FUNCTION_BLOCK ChangeDetect (* Ground-truth reference: fires CHG only when the REAL input value actually changed *)
  (* Standard: 61499-2; Description: Educational reference, ported for the Meisterschulen am Ostbahnhof IEC 61499 training repository. Original design (c) nxtControl GmbH, from the UniversalAutomation.org 'IEC 61499: primer course' curriculum exercise Final.sln (also present in the LiftingLuggage_*.sln/Starter.sln exercises), IEC61499/ChangeDetect.fbt - included here under the same educational-use terms as the rest of that curriculum. This port: Copyright (c) 2026 Meisterschulen am Ostbahnhof, EPL-2.0, https://www.eclipse.org/legal/epl-2.0/ *)
  (* Version 0.0, 2016-05-28, Andrei, nxtControl GmbH, Original EAE/nxtControl design (Template), source: Final.sln (identical copies in LiftingLuggage_*.sln, Starter.sln) *)
  (* Version 1.0, 2026-09-03, Franz Höpfinger, Meisterschulen am Ostbahnhof, Ported from EAE/nxtControl format (LibraryElement.dtd, ST as an attribute with escapes) to 4diac's FBType XSD (ST as CDATA). Interface, ECC, and both algorithms otherwise unchanged. Part of the CylinderH continuous-simulation reference - see ContinuousCylinderSimulation.md *)
  PACKAGE Meins::DesingPatterns::ContinuousCylinderSimulation;
  (* Documentation:
  Ground-truth reference, not a Vyatkin Module 6 slide pattern. Simple REAL change-detection filter, ported as-is from the UniversalAutomation.org "IEC 61499: primer course" curriculum (Final.sln, IEC61499/ChangeDetect.fbt, original format: EAE/nxtControl LibraryElement.dtd). Used by CylinderHCore.fbt in this folder to throttle the integrator's continuous out value down to only the moments it actually changes, before reporting the cylinder's Position onward.
  *)
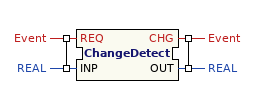
  EVENT_INPUT
    REQ WITH INP; (* Normal Execution Request *)
  END_EVENT
  EVENT_OUTPUT
    CHG WITH OUT; (* Execution Confirmation: fired every REQ, but only carries a new value on an actual change *)
  END_EVENT
  VAR_INPUT
    INP : REAL;
  END_VAR
  VAR_OUTPUT
    OUT : REAL;
  END_VAR
  VAR
    PREV : REAL; (* Value seen on the previous REQ *)
  END_VAR
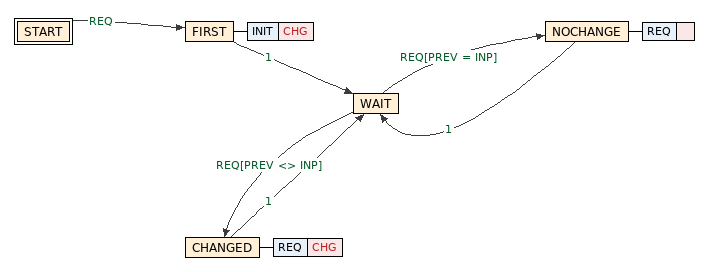
  EC_STATES
    START; (* Initial State *)
    FIRST : INIT -> CHG; (* First REQ ever received: always report it *)
    WAIT; (* Waiting for the next REQ *)
    NOCHANGE : REQ; (* Value unchanged: stay quiet *)
    CHANGED : REQ -> CHG; (* Value changed: report it *)
  END_STATES
  EC_TRANSITIONS
    START TO FIRST := REQ;
    FIRST TO WAIT := 1;
    WAIT TO NOCHANGE := REQ[PREV = INP];
    NOCHANGE TO WAIT := 1;
    WAIT TO CHANGED := REQ[PREV <> INP];
    CHANGED TO WAIT := 1;
  END_TRANSITIONS
  ALGORITHM INIT IN ST: (* First value ever seen: store and report it *)
PREV := INP;
OUT := INP;
  END_ALGORITHM
  ALGORITHM REQ IN ST: (* Store the current value; OUT is only meaningful when this state also fires CHG *)
PREV := INP;
OUT := INP;
  END_ALGORITHM
END_FUNCTION_BLOCK
